(* PLC project io_single_acting_valve, Dassault Systèmes ControlBuild 2024x *)
(* stored: creationDateTime 2023-10-03T11:12:49-01:00 *)

PROGRAM panel
  VAR_OUTPUT
    openValvePB : BOOL := false;
  END_VAR

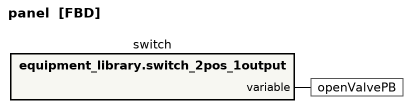
(* FBD diagram, written out as Structured Text *)
switch();
openValvePB := switch.variable;
END_PROGRAM

(* Integrated object C/C+OP of a single acting valve *)
PROGRAM io_library.io_single_acting_valve
  VAR_INPUT
    acknowledgePB : BOOL := false;
  END_VAR
  VAR_INPUT
    autoMode : BOOL := false;
    manualMode : BOOL := false;
  END_VAR
  VAR_INPUT
    autoOpenCmd : BOOL := false;
  END_VAR
  VAR_INPUT
    inputFlow : REAL := 0.0;
  END_VAR
  VAR_OUTPUT
    openedSensor : BOOL := false;
    closedSensor : BOOL := false;
  END_VAR
  VAR_OUTPUT
    generalFault : BOOL := false;
    outputFlow : REAL := 0.0;
    percentOpening : REAL := 0.0;
  END_VAR

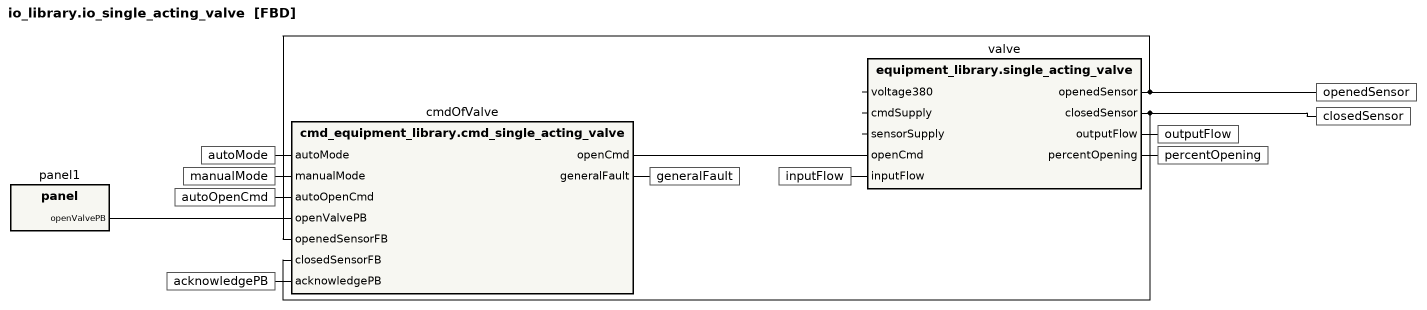
(* FBD diagram, written out as Structured Text *)
panel1();
cmdOfValve(autoMode := autoMode, manualMode := manualMode, autoOpenCmd := autoOpenCmd, openValvePB := panel1.openValvePB, openedSensorFB := valve.openedSensor, closedSensorFB := valve.closedSensor, acknowledgePB := acknowledgePB);
valve(openCmd := cmdOfValve.openCmd, inputFlow := inputFlow);
openedSensor := valve.openedSensor;
closedSensor := valve.closedSensor;
outputFlow := valve.outputFlow;
percentOpening := valve.percentOpening;
generalFault := cmdOfValve.generalFault;
END_PROGRAM
